PROGRAM P_MBus_Fast
VAR
	fbMBUSKL6781		: FB_MBUSKL6781;
END_VAR

fbMBUSKL6781(
	usiRetries	:= , 
	bStart		:= , 
	bDisabled	:= , 
	bBusy		=> , 
	bReady		=> , 
	bError		=> , 
	eError		=> , 
	stComIn		:= GVL_IO.stComIn, 
	stComOut	:= GVL_IO.stComOut, 
	stCom		:= GVL_IO.stCom);

END_PROGRAM

(* stored: Version 1.1.0.1, ProductVersion 3.1.4024.6
   POU P_MBus_Fast: Id {503c5f3f-a6e9-4d4d-84bc-c417aab4f4ba}, SpecialFunc None *)
